# EPICS autosave request: apps/svtIntlkApp/Db/svtIntlk_settings.req
file svtIntlk.req P=HPS_INTLK:SVT_SUP:
file svtIntlk.req P=HPS_INTLK:SVT_RTN:
file svtIntlk.req P=HPS_INTLK:FE_SUP:
file svtIntlk.req P=HPS_INTLK:FE_RTN:
file svtIntlk.req P=HPS_INTLK:DET_VAC:
